TYPE ST_JoystickInputScaling :
STRUCT
	fMaxInputValue : LREAL;
	fMinInputValue : LREAL;
	fNeutralInputValue : LREAL;
	fNeutralDeadband : LREAL;
	fMaxOutputValue : LREAL;
	fMinOutputValue : LREAL;
	fNeutralOutputValue : LREAL;
END_STRUCT
END_TYPE

(* stored: Version 1.1.0.1, ProductVersion 3.1.4024.12
   DUT ST_JoystickInputScaling: Id {3ef35e61-e42a-4299-824a-51fccff0c0d4} *)
